// TIA Portal V18 export
DATA_BLOCK "AHUAI"   // DB111
{ S7_Optimized_Access := 'FALSE' }
VERSION : 0.1
// stored: AutoNumber false, DBAccessibleFromOPCUA true, IsOnlyStoredInLoadMemory false, IsWriteProtectedInAS false
   VAR
      AI { S7_SetPoint := 'True'} : "UDT_AHUsAI";
   END_VAR
BEGIN
   AI.rIAQ[1..3] := 0.0;
   AI.rBuildingdP[1..3] := 0.0;
   AI.rRoomAirTemp_PLC_AI[1..3] := 0.0;
   AI.rSupplyAirTemp[1] := 26.69;
   AI.rSupplyAirTemp[2] := 0.0;
   AI.rSupplyAirTemp[3] := 22.39;
   AI.rReturnAirTemp[1..3] := 0.0;
   AI.rFrostProtWaterTemp[1] := 3276.7;
   AI.rFrostProtWaterTemp[2] := 0.0;
   AI.rFrostProtWaterTemp[3] := 21.31;
   AI.rFrostProtAirTemp[1] := 17.07954;
   AI.rFrostProtAirTemp[2..3] := 0.0;
   AI.rRoomAirRelHumi[1..2] := 0.0;
   AI.rRoomAirRelHumi[3] := 21.23;
   AI.rReserve[1..3] := 0.0;
   AI.rSAFilterdP[1] := 5.714699;
   AI.rSAFilterdP[2..3] := 0.0;
   AI.cRoomTempSelect[1] := 2;
END_DATA_BLOCK
